(* LS Electric XG5000 project: XEM_Motion_Demo *)
(* PLC LSPLC *)
(* module base 0 slot 0: Input/Output Module:XEM-DN/DP32HP (DC 24V Input, Transistor Output, 32 Contacts) *)
(* module base 0 slot 1: Internal Positioning:XBF-PO06E (Open Collector Type, 6 Axis) *)
VAR_GLOBAL
    Axis1_Command : Motion_Command_type; (* Commands for Axis 1 *)
    Axis1_Status : Motion_Status_type; (* Status for axis 1 *)
    Axis2_Command : Motion_Command_type; (* Commands for Axis 2 *)
    Axis2_Status : Motion_Status_type; (* Status for axis 2 *)
    Axis3_Command : Motion_Command_type; (* Commands for Axis 3 *)
    Axis3_Status : Motion_Status_type; (* Status for axis 3 *)
    Reset_Servo_Errors : BOOL; (* Acknowledge servo errors *)
    Turn_On_Servos : BOOL; (* Command to turn on all the servos *)
END_VAR

TYPE Motion_Command_type : (* contains motion commands and data for those commands *)
STRUCT
    Servo_On : BOOL; (* Command to turn servo on *)
    Home : BOOL; (* command to home axis *)
    Direct_Absolute_Move : BOOL; (* command for direct start absolute move *)
    Direct_Relative_Move : BOOL; (* command for direct start relative move *)
    Direct_Feed_Move : BOOL; (* command to perform a direct start feed move *)
    Direct_Speed_Move : BOOL; (* command to run axis direct start speed control. *)
    Indirect_Absolute_Move : BOOL; (* command for indirect start absolute move *)
    Indirect_Relative_Move : BOOL; (* command for indirect start relative move *)
    Indirect_Feed_Move : BOOL; (* command for indirect start feed move *)
    Indirect_Speed_Move : BOOL; (* command for indirect start speed control. *)
    Linear_Interpolation_Move : BOOL; (* command for indirect start for linear interpolation move *)
    Cirular_Interpolation_Start : BOOL; (* command for indirect start of circular interpolation move *)
    Helical_Interpolation_Start : BOOL; (* command for indirect start of helical interpolation move *)
    Ellipse_Interpolation_Start : BOOL; (* command to start ellipse interpolation. *)
    Stop_Axis : BOOL; (* perform a deceleration stop *)
    EStop_Axis : BOOL; (* peform an emergency stop *)
    Reset_Axis_Error : BOOL; (* reset an axis error *)
    Target_Position : DINT; (* target position for direct start moves in pulses *)
    Target_Speed : UDINT; (* target speed for direct start moves in pulses/sec *)
    Dwell_Time : UINT; (* dwell time in milliseconds *)
    Accel_Selection : USINT; (* Acceleration setting in XG-PM settings to use. *)
    Decel_Selection : USINT; (* Deceleration setting in XG-PM settings to use *)
END_STRUCT;
END_TYPE

TYPE Motion_Status_type : (* Motion status information *)
STRUCT
    Axis_Ready : BOOL; (* axis is ready for commands *)
    Busy : BOOL; (* status that the axis is busy *)
    Error_Present : BOOL; (* status of an error *)
    Move_Done : BOOL; (* status that move is done *)
    Homed : BOOL; (* status that axis is homed. *)
    Current_Position_Pulses : DINT; (* Current position of the axis in pulses *)
    Current_Speed_Pulses : DINT; (* Current speed of the axis in pulses *)
    Current_Torque : INT; (* current torque *)
    Error_Number : UINT; (* current error number *)
    Commanded_Position : DINT; (* commanded position *)
    Commanded_Speed : DINT; (* commanded speed *)
    Current_Step_Number : UINT; (* current step number of the operation being performed *)
    State1 : ARRAY[0..7] OF BOOL; (* array for state 1 of Axis state fb *)
    State2 : ARRAY[0..7] OF BOOL; (* array for state 2 of Axis state fb *)
    State3 : ARRAY[0..7] OF BOOL; (* array for state 3 of Axis state fb *)
    State4 : ARRAY[0..7] OF BOOL; (* array for state 4 of Axis state fb *)
    State5 : ARRAY[0..7] OF BOOL; (* array for state 5 of Axis state fb *)
    State6 : ARRAY[0..7] OF BOOL; (* array for state 6 of Axis state fb *)
    State7 : ARRAY[0..7] OF BOOL; (* array for state 7 of Axis state fb *)
    Servo_Drive_Ready : BOOL; (* status that the servo drive being controlled is ready *)
    Servo_Drive_Error : BOOL; (* Status that the servo drive being controlled doesn't have an error *)
END_STRUCT;
END_TYPE

PROGRAM Interpolation_Routines (* task: Scan Program *)
(* control the demo code for interpolation movements *)
VAR
    Axes_Are_Homed : BOOL; (* status that the 3 axes are homed *)
    Axes_Are_Ready : BOOL; (* status command that axes 1 thru 3 are ready *)
    Home_Axes : BOOL; (* home all the axes *)
    Motion_Manager_State : USINT := 0; (* State machine variable for motion manager *)
    Run_Circular_Interpolation : BOOL := 0; (* command to run circular interpolation demo *)
    Run_Ellipse_Interpolation : BOOL := 0; (* Command to run ellipse interpolation demo *)
    Run_Helical_Interpolation : BOOL := 0; (* command to run helical interpolation demo *)
    Run_Linear_Interpolation : BOOL := 0; (* command to run linear interpolation demo *)
    TempInt : INT;
    TempWord : WORD := 60502;
END_VAR
VAR_EXTERNAL
    Axis1_Command : Motion_Command_type; (* Commands for Axis 1 *)
    Axis1_Status : Motion_Status_type; (* Status for axis 1 *)
    Axis2_Command : Motion_Command_type; (* Commands for Axis 2 *)
    Axis2_Status : Motion_Status_type; (* Status for axis 2 *)
    Axis3_Command : Motion_Command_type; (* Commands for Axis 3 *)
    Axis3_Status : Motion_Status_type; (* Status for axis 3 *)
    Turn_On_Servos : BOOL; (* Command to turn on all the servos *)
END_VAR
(* 
AutomationDirect.com has provided this code for convenience. This sample code is provided "as-is" with no expressed or implied warranty. 
 If the end user includes any of the sample code (in whole or part), it is the user's responsibility to completely modify, integrate, and test any code to ensure it meets all system and 
 safety requirements for the intended application or system.
 *)


//Make sure axes are ready for commands
IF (Axis1_Status.Axis_Ready AND Axis2_Status.Axis_Ready AND Axis3_Status.Axis_Ready) AND (Axis1_Status.Busy = FALSE) AND (Axis2_Status.Busy = FALSE) AND (Axis3_Status.Busy = FALSE) THEN
	Axes_Are_Ready := TRUE;
ELSE
	Axes_Are_Ready := FALSE;

END_IF;
	
//make sure Axes are homed
IF Axis1_Status.Homed AND Axis2_Status.Homed AND Axis3_Status.Homed THEN
	Axes_Are_Homed := TRUE;
ELSE	
	Axes_Are_Homed := FALSE;
	
END_IF;

//Reset State machine if there is a drive alarm or the servos are turned off.
IF (%IX0.0.11 = FALSE) OR (Turn_On_Servos = FALSE) THEN
	Motion_Manager_State := 0;
END_IF;

(* State machine for running the three interpolation demos.  It will move axes to starting positions using the direct start commands of those axes. *)
CASE Motion_Manager_State OF
	
	//wait for command to run a demo.
	0:
		Axis1_Command.Direct_Absolute_Move := FALSE;
		Axis2_Command.Direct_Absolute_Move := FALSE;
		Axis3_Command.Direct_Absolute_Move := FALSE;
		
		//home axes 
		IF Axes_Are_Ready AND Home_Axes THEN
			Home_Axes := FALSE;
			Motion_Manager_State := 100;
			
		//Allow interpolation commands if axes are ready and homed.  They use absolute movements to go to starting positions	
		ELSIF Axes_Are_Ready AND Axes_Are_Homed THEN
			
				IF (Run_Linear_Interpolation = TRUE) THEN
					Run_Linear_Interpolation := FALSE;
					Motion_Manager_State := 10;
				
				ELSIF(Run_Circular_Interpolation = TRUE) THEN
					Run_Circular_Interpolation := FALSE;
					Motion_Manager_State := 20;
					
				ELSIF(Run_Helical_Interpolation = TRUE) THEN
					Run_Helical_Interpolation := FALSE;
					Motion_Manager_State := 30;		
					
				ELSIF(Run_Ellipse_Interpolation = TRUE) THEN
					Run_Ellipse_Interpolation := FALSE;
					Motion_Manager_State := 40;	
						
				END_IF;	

		
		//Reset Interpolation commands if axes are not ready
		ELSE	
				Run_Helical_Interpolation := FALSE;
				Run_Circular_Interpolation := FALSE;
				Run_Linear_Interpolation := FALSE;
		END_IF;
	
	
	(**********************
	     Peform Linear interpolation.
	     ***************************) 
	// Move Axis 3(z on gantry) up so that Axis 1(x) and Axis 2(y) can be moved to starting position.			
	10:	
		IF (Axis3_Status.Current_Position_Pulses = 200)  THEN
			Motion_Manager_State := 11;
			
		ELSE	
			Axis3_Command.Target_Position :=  200;
			Axis3_Command.Target_Speed := 500;
			
			Axis3_Command.Direct_Absolute_Move := TRUE;
			
			IF(Axis3_Status.Current_Position_Pulses = 200) THEN
				Axis3_Command.Direct_Absolute_Move := FALSE;
				Motion_Manager_State := 11;
			END_IF;
			
		END_IF;	
		
	//Axis 1 (x) and Axis 2(y) can move to linear interpolation start position	
	11: 
		Axis1_Command.Target_Position :=  200;
		Axis1_Command.Target_Speed := 500;		
			
		Axis2_Command.Target_Position :=  200;
		Axis2_Command.Target_Speed := 500;
		
		Axis1_Command.Direct_Absolute_Move := TRUE;
		Axis2_Command.Direct_Absolute_Move := TRUE;
	
		
		IF (Axis1_Status.Current_Position_Pulses = 200)  AND (Axis2_Status.Current_Position_Pulses = 200) THEN
			Axis1_Command.Direct_Absolute_Move := FALSE;
			Axis2_Command.Direct_Absolute_Move := FALSE;
			Axis3_Command.Direct_Absolute_Move := FALSE;
			Motion_Manager_State := 12;
		END_IF;	
		
	// Move Axis 3 (z) to 0 position so pen is touching paper	
	12:	
		Axis3_Command.Target_Position :=  0;
		Axis3_Command.Target_Speed := 500;
		
		Axis3_Command.Direct_Absolute_Move := TRUE;
	
		
		IF(Axis3_Status.Current_Position_Pulses = 0) THEN
			Axis3_Command.Direct_Absolute_Move := FALSE;
			Motion_Manager_State := 13;
		END_IF;

	//Start linear interpolation command. Axis 1 is master so it is the only XPM_IST that needs to be run
	13:
		IF Axis1_Status.Axis_Ready AND Axis2_Status.Axis_Ready THEN
			Axis1_Command.Linear_Interpolation_Move := TRUE;
		END_IF;	
		
	 	IF (Axis1_Status.Busy = TRUE)  AND (Axis2_Status.Busy = TRUE) THEN
			Motion_Manager_State := 14;
		END_IF;	
		
	//wait for interpolation to be done then go back to wait for command state	
	14:
		IF Axis1_Status.Move_Done AND Axis2_Status.Move_Done THEN
			Motion_Manager_State := 15;
		END_IF;
		
	//Move the axes to a wait position	 for states 15 and 16
	15:	
			Axis3_Command.Target_Position :=  200;
			Axis3_Command.Target_Speed := 500;			
			Axis3_Command.Direct_Absolute_Move := TRUE;
			
			IF(Axis3_Status.Current_Position_Pulses = 200) THEN
				Axis3_Command.Direct_Absolute_Move := FALSE;
				Motion_Manager_State := 16;
			END_IF;
		
	16:
		Axis1_Command.Target_Position :=  0;
		Axis1_Command.Target_Speed := 500;		
			
		Axis2_Command.Target_Position :=  0;
		Axis2_Command.Target_Speed := 500;
		
		Axis1_Command.Direct_Absolute_Move := TRUE;
		Axis2_Command.Direct_Absolute_Move := TRUE;		
	
		IF (Axis1_Status.Current_Position_Pulses = 0)  AND (Axis2_Status.Current_Position_Pulses = 0) THEN
			Axis1_Command.Direct_Absolute_Move := FALSE;
			Axis2_Command.Direct_Absolute_Move := FALSE;
			Axis3_Command.Direct_Absolute_Move := FALSE;
			Motion_Manager_State := 0;
		END_IF;	
	
	
	(******************************
		 Peform Circular interpolation. 
		 **********************)
	 //MOVE Axis 3(z on gantry) up so that Axis 1(x) and Axis 2(y) can be moved to starting position.			
	20:	
		
		IF (Axis3_Status.Current_Position_Pulses = 200)   THEN
			Motion_Manager_State := 21;
			
		ELSE	
			Axis3_Command.Target_Position :=  200;
			Axis3_Command.Target_Speed := 500;
			
			Axis3_Command.Direct_Absolute_Move := TRUE;
			
			IF(Axis3_Status.Current_Position_Pulses = 200) THEN
				Axis3_Command.Direct_Absolute_Move := FALSE;
				Motion_Manager_State := 21;
			END_IF;
			
		END_IF;	
		
	// Axis 1 (x) and Axis 2(y) can move to circular interpolation start position	
	21: 
		Axis1_Command.Target_Position :=  200;
		Axis1_Command.Target_Speed := 500;		
			
		Axis2_Command.Target_Position :=  1500;
		Axis2_Command.Target_Speed := 500;
		
		Axis1_Command.Direct_Absolute_Move := TRUE;
		Axis2_Command.Direct_Absolute_Move := TRUE;
	
		
		IF (Axis1_Status.Current_Position_Pulses = 200)  AND (Axis2_Status.Current_Position_Pulses = 1500) THEN
			Axis1_Command.Direct_Absolute_Move := FALSE;
			Axis2_Command.Direct_Absolute_Move := FALSE;
			Axis3_Command.Direct_Absolute_Move := FALSE;
			Motion_Manager_State := 22;
		END_IF;	
		
	// move Axis 3 (z) to 0 position so pen is touching paper	
	22:	
		Axis3_Command.Target_Position :=  0;
		Axis3_Command.Target_Speed := 500;
		
		Axis3_Command.Direct_Absolute_Move := TRUE;
	
		
		IF(Axis3_Status.Current_Position_Pulses = 0) THEN
			Axis3_Command.Direct_Absolute_Move := FALSE;
			Motion_Manager_State := 23;
		END_IF;
	
	//Start Circular interpolation command. Axis 1 is master so it is the only XPM_IST that needs to be run
	23:
		IF Axis1_Status.Axis_Ready AND Axis2_Status.Axis_Ready THEN
			Axis1_Command.Cirular_Interpolation_Start := TRUE;
		END_IF;	

	 	IF (Axis1_Status.Busy = TRUE)  AND (Axis2_Status.Busy = TRUE) THEN
			Motion_Manager_State := 24;
		END_IF;			
	
	//wait for interpolation to be done 
	24:
		IF Axis1_Status.Move_Done AND Axis2_Status.Move_Done THEN
			Motion_Manager_State := 25;
		END_IF;	
	
		//Move the axes to a wait position	 for states 25 and 26
	25:	
			Axis3_Command.Target_Position :=  200;
			Axis3_Command.Target_Speed := 500;			
			Axis3_Command.Direct_Absolute_Move := TRUE;
			
			IF(Axis3_Status.Current_Position_Pulses = 200) THEN
				Axis3_Command.Direct_Absolute_Move := FALSE;
				Motion_Manager_State := 26;
			END_IF;
		
	26:
		Axis1_Command.Target_Position :=  0;
		Axis1_Command.Target_Speed := 500;		
			
		Axis2_Command.Target_Position :=  0;
		Axis2_Command.Target_Speed := 500;
		
		Axis1_Command.Direct_Absolute_Move := TRUE;
		Axis2_Command.Direct_Absolute_Move := TRUE;		
	
		IF (Axis1_Status.Current_Position_Pulses = 0)  AND (Axis2_Status.Current_Position_Pulses = 0) THEN
			Axis1_Command.Direct_Absolute_Move := FALSE;
			Axis2_Command.Direct_Absolute_Move := FALSE;
			Axis3_Command.Direct_Absolute_Move := FALSE;
			Motion_Manager_State := 0;
		END_IF;	
	
	
(******************************
		 Peform Helical interpolation. 
		 **********************)
	 //MOVE Axis 3(z on gantry) up so that Axis 1(x) and Axis 2(y) can be moved to starting position.			
	30:	
		
		IF (Axis3_Status.Current_Position_Pulses = 200)   THEN
			Motion_Manager_State := 31;
			
		ELSE	
			Axis3_Command.Target_Position :=  200;
			Axis3_Command.Target_Speed := 500;
			
			Axis3_Command.Direct_Absolute_Move := TRUE;
			
			IF(Axis3_Status.Current_Position_Pulses = 200) THEN
				Axis3_Command.Direct_Absolute_Move := FALSE;
				Motion_Manager_State := 31;
			END_IF;
			
		END_IF;	
		
	// Axis 1 (x) and Axis 2(y) can move to helical interpolation start position	
	31: 
		Axis1_Command.Target_Position :=  600;
		Axis1_Command.Target_Speed := 500;		
			
		Axis2_Command.Target_Position :=  400;
		Axis2_Command.Target_Speed := 500;
		
		Axis1_Command.Direct_Absolute_Move := TRUE;
		Axis2_Command.Direct_Absolute_Move := TRUE;
	
		
		IF (Axis1_Status.Current_Position_Pulses = 600)  AND (Axis2_Status.Current_Position_Pulses = 400) THEN
			Axis1_Command.Direct_Absolute_Move := FALSE;
			Axis2_Command.Direct_Absolute_Move := FALSE;
			Axis3_Command.Direct_Absolute_Move := FALSE;
			Motion_Manager_State := 32;
		END_IF;	
		
	// move Axis 3 (z) to 0 position so pen is touching paper	
	32:	
		Axis3_Command.Target_Position :=  0;
		Axis3_Command.Target_Speed := 500;
		
		Axis3_Command.Direct_Absolute_Move := TRUE;
	
		
		IF(Axis3_Status.Current_Position_Pulses = 0) THEN
			Axis3_Command.Direct_Absolute_Move := FALSE;
			Motion_Manager_State := 33;
		END_IF;
	
	//Start Helical interpolation command. Axis 1 is master so it is the only XPM_IST that needs to be run
	33:
		IF Axis1_Status.Axis_Ready AND Axis2_Status.Axis_Ready AND Axis3_Status.Axis_Ready THEN
			Axis1_Command.Helical_Interpolation_Start := TRUE;
		END_IF;	

	 	IF (Axis1_Status.Busy = TRUE)  AND (Axis2_Status.Busy = TRUE) AND (Axis3_Status.Busy = TRUE) THEN
			Motion_Manager_State := 34;
		END_IF;	
		
	//wait for interpolation to be done 
	34:
		IF Axis1_Status.Move_Done AND Axis2_Status.Move_Done THEN
			Motion_Manager_State := 35;
		END_IF;	
	
		//Move the axes to a wait position for states 35 and 36
	35:	
			Axis3_Command.Target_Position :=  200;
			Axis3_Command.Target_Speed := 500;			
			Axis3_Command.Direct_Absolute_Move := TRUE;
			
			IF(Axis3_Status.Current_Position_Pulses = 200) THEN
				Axis3_Command.Direct_Absolute_Move := FALSE;
				Motion_Manager_State := 36;
			END_IF;
		
	36:
		Axis1_Command.Target_Position :=  0;
		Axis1_Command.Target_Speed := 100;		
			
		Axis2_Command.Target_Position :=  0;
		Axis2_Command.Target_Speed := 500;
		
		Axis1_Command.Direct_Absolute_Move := TRUE;
		Axis2_Command.Direct_Absolute_Move := TRUE;		
	
		IF (Axis1_Status.Current_Position_Pulses = 0)  AND (Axis2_Status.Current_Position_Pulses = 0) THEN
			Axis1_Command.Direct_Absolute_Move := FALSE;
			Axis2_Command.Direct_Absolute_Move := FALSE;
			Axis3_Command.Direct_Absolute_Move := FALSE;
			Motion_Manager_State := 0;
		END_IF;		
	
	
	
(******************************
		 Peform Ellipse interpolation. 
		 **********************)
	 //MOVE Axis 3(z on gantry) up so that Axis 1(x) and Axis 2(y) can be moved to starting position.			
	40:	
		
		IF (Axis3_Status.Current_Position_Pulses = 200)   THEN
			Motion_Manager_State := 41;
			
		ELSE	
			Axis3_Command.Target_Position :=  200;
			Axis3_Command.Target_Speed := 500;
			
			Axis3_Command.Direct_Absolute_Move := TRUE;
			
			IF(Axis3_Status.Current_Position_Pulses = 200) THEN
				Axis3_Command.Direct_Absolute_Move := FALSE;
				Motion_Manager_State := 41;
			END_IF;
			
		END_IF;	
		
	//Axis 1 (x) and Axis 2(y) can move to ellipse interpolation start position	
	41: 
		Axis1_Command.Target_Position :=  0;
		Axis1_Command.Target_Speed := 500;		
			
		Axis2_Command.Target_Position :=  0;
		Axis2_Command.Target_Speed := 500;
		
		Axis1_Command.Direct_Absolute_Move := TRUE;
		Axis2_Command.Direct_Absolute_Move := TRUE;
	
		
		IF (Axis1_Status.Current_Position_Pulses = 0)  AND (Axis2_Status.Current_Position_Pulses = 0) THEN
			Axis1_Command.Direct_Absolute_Move := FALSE;
			Axis2_Command.Direct_Absolute_Move := FALSE;
			Axis3_Command.Direct_Absolute_Move := FALSE;
			Motion_Manager_State := 42;
		END_IF;	
		
	// move Axis 3 (z) to 0 position so pen is touching paper	
	42:	
		Axis3_Command.Target_Position :=  0;
		Axis3_Command.Target_Speed := 500;
		
		Axis3_Command.Direct_Absolute_Move := TRUE;
	
		
		IF(Axis3_Status.Current_Position_Pulses = 0) THEN
			Axis3_Command.Direct_Absolute_Move := FALSE;
			Motion_Manager_State := 43;
		END_IF;
	
	//Start Ellipse interpolation command. Axis 1 is master so it is the only XPM_ELIN that needs to be run
	43:
		IF Axis1_Status.Axis_Ready AND Axis2_Status.Axis_Ready THEN
			Axis1_Command.Ellipse_Interpolation_Start := TRUE;
		END_IF;	

	 	IF (Axis1_Status.Busy = TRUE)  AND (Axis2_Status.Busy = TRUE) THEN
			Motion_Manager_State := 44;
		END_IF;			
	
	//wait for interpolation to be done 
	44:
		IF Axis1_Status.Move_Done AND Axis2_Status.Move_Done THEN
			Motion_Manager_State := 45;
		END_IF;	
	
		//Move the axes to a wait position	 for states 45 and 46
	45:	
			Axis3_Command.Target_Position :=  200;
			Axis3_Command.Target_Speed := 500;			
			Axis3_Command.Direct_Absolute_Move := TRUE;
			
			IF(Axis3_Status.Current_Position_Pulses = 200) THEN
				Axis3_Command.Direct_Absolute_Move := FALSE;
				Motion_Manager_State := 46;
			END_IF;
		
	46:
		Axis1_Command.Target_Position :=  0;
		Axis1_Command.Target_Speed := 500;		
			
		Axis2_Command.Target_Position :=  0;
		Axis2_Command.Target_Speed := 500;
		
		Axis1_Command.Direct_Absolute_Move := TRUE;
		Axis2_Command.Direct_Absolute_Move := TRUE;		
	
		IF (Axis1_Status.Current_Position_Pulses = 0)  AND (Axis2_Status.Current_Position_Pulses = 0) THEN
			Axis1_Command.Direct_Absolute_Move := FALSE;
			Axis2_Command.Direct_Absolute_Move := FALSE;
			Axis3_Command.Direct_Absolute_Move := FALSE;
			Motion_Manager_State := 0;
		END_IF;		
	
	
	
	
	//home axes
	100:
		Axis1_Command.Home := TRUE;
		Axis2_Command.Home := TRUE;
		
		IF (Axis1_Status.Homed AND Axis2_Status.Homed) THEN
			Motion_Manager_State := 101;
		END_IF;
	
	//Home Axis 3 separately so the pen doesn't drag on the surface.
	101:
		Axis3_Command.Home := TRUE;
	
		IF (Axis3_Status.Homed) THEN
			Motion_Manager_State := 102;
		END_IF;
 
	//move Axis 3 to a wait position so Pen isn't constantly in contact with the surface
	102:	
			Axis3_Command.Target_Position :=  200;
			Axis3_Command.Target_Speed := 500;			
			Axis3_Command.Direct_Absolute_Move := TRUE;
			
			IF(Axis3_Status.Current_Position_Pulses = 200) THEN
				Axis3_Command.Direct_Absolute_Move := FALSE;
				Motion_Manager_State := 0;
			END_IF;
		
		
END_CASE;
END_PROGRAM

PROGRAM Axis1_Motion_Program (* task: Scan Program *)
(* program for XPM function blocks that perform actions for axis 1 *)
VAR_EXTERNAL
    Axis1_Command : Motion_Command_type; (* Commands for Axis 1 *)
    Axis1_Status : Motion_Status_type; (* Status for axis 1 *)
END_VAR
VAR
    Axis_State_FB : XPM_SRD; (* Axis state function block *)
    Axis_Status_FB : XPM_CRD; (* Axis status function block *)
    CurPos_Conversion_Value : REAL; (* value to convert pulse position to engineering unit position *)
    Deceleration_Stop_FB : XPM_STP; (* function block for deceleration stop *)
    DirectStart_ABS_INC : BOOL; (* False - Absolute Positioning;  True -  Relative Positioning *)
    DirectStart_Control : USINT; (* Control Method for Direct Start.  0 - Position Control; 1 - Speed Control;  2 - FEED Control *)
    Direct_Start_FB : XPM_DST; (* function block for direct start commands *)
    Emergency_Stop_FB : XPM_EMG; (* function block to perform emergency stop *)
    Error_Reset_FB : XPM_RST; (* function block for resetting axis error *)
    Home_FB : XPM_ORG; (* function block to home axis *)
    Indirect_Start_FB : XPM_IST; (* function block to perform indirect start procedures *)
    Indirect_Step_Number : UINT; (* Step number for Indirect movement *)
    TempR1 : REAL; (* temporary real storage *)
    TempR2 : REAL; (* temporary real storage *)
    XPM_ELIN_INST : XPM_ELIN;
END_VAR
VAR
    _e1 : R_TRIG;
    _e2 : R_TRIG;
    _e3 : R_TRIG;
    _e4 : R_TRIG;
    _e5 : R_TRIG;
    _e6 : R_TRIG;
    _e7 : R_TRIG;
    _e8 : R_TRIG;
    _e9 : R_TRIG;
    _e10 : R_TRIG;
    _e11 : R_TRIG;
    _e12 : R_TRIG;
    _e13 : R_TRIG;
    _e14 : R_TRIG;
    _e15 : R_TRIG;
END_VAR

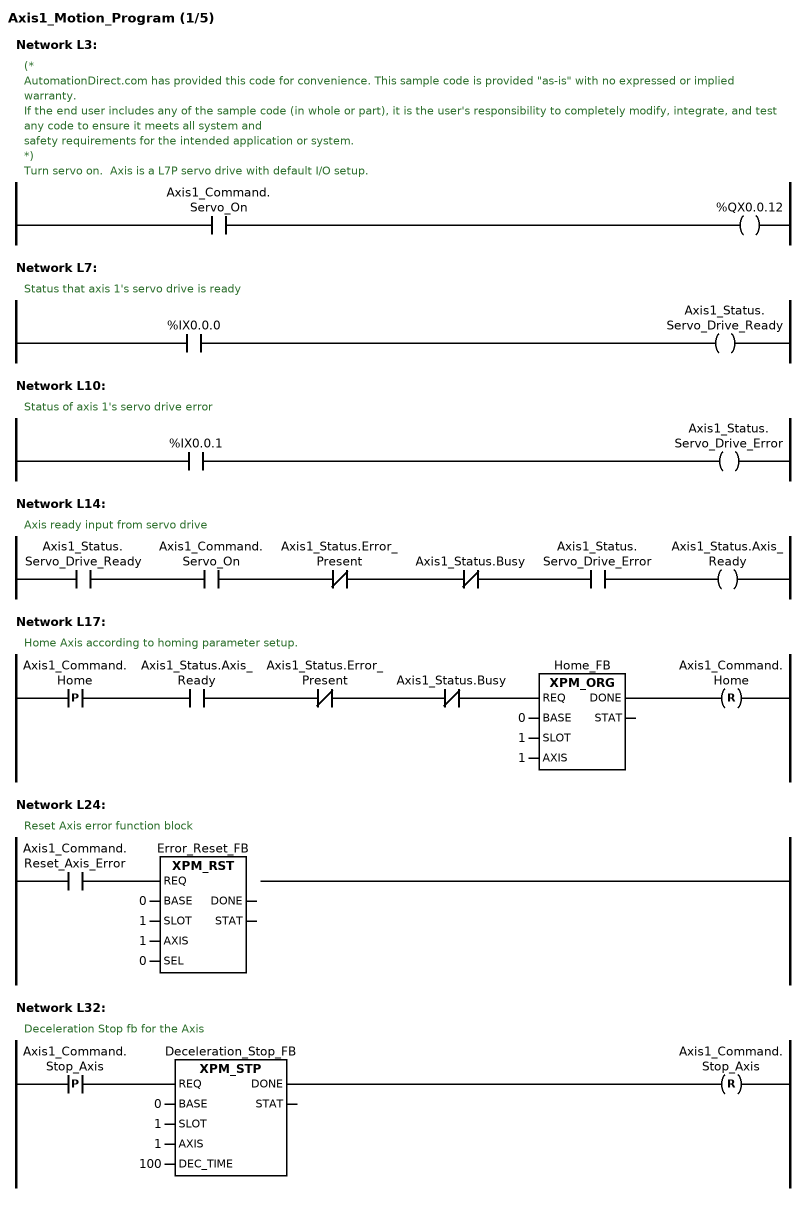
(* ( * / AutomationDirect.com has provided this code for convenience. This sample code is provided "as-is" with no expressed or implied warranty. / If the end user includes any of the sample code (in whole or part), it is the user's responsibility to completely modify, integrate, and test any code to ensure it meets all system and / safety requirements for the intended application or system. / * ) *)
(* Turn servo on.  Axis is a L7P servo drive with default I/O setup. *)
(* Rung L3 *)
%QX0.0.12 := Axis1_Command.Servo_On;
(* Status that axis 1's servo drive is ready *)
(* Rung L7 *)
Axis1_Status.Servo_Drive_Ready := %IX0.0.0;
(* Status of axis 1's servo drive error *)
(* Rung L10 *)
Axis1_Status.Servo_Drive_Error := %IX0.0.1;
(* Axis ready input from servo drive *)
(* Rung L14 *)
Axis1_Status.Axis_Ready := Axis1_Status.Servo_Drive_Ready AND Axis1_Command.Servo_On AND NOT Axis1_Status.Error_Present AND NOT Axis1_Status.Busy AND Axis1_Status.Servo_Drive_Error;
(* Home Axis according to homing parameter setup. *)
(* Rung L17 *)
_e1(CLK := Axis1_Command.Home);
Home_FB(REQ := _e1.Q AND Axis1_Status.Axis_Ready AND NOT Axis1_Status.Error_Present AND NOT Axis1_Status.Busy, BASE := 0, SLOT := 1, AXIS := 1);
IF Home_FB.DONE THEN Axis1_Command.Home := FALSE; END_IF;
(* Reset Axis error function block *)
(* Rung L24 *)
Error_Reset_FB(REQ := Axis1_Command.Reset_Axis_Error, BASE := 0, SLOT := 1, AXIS := 1, SEL := 0);
(* Deceleration Stop fb for the Axis *)
(* Rung L32 *)
_e2(CLK := Axis1_Command.Stop_Axis);
Deceleration_Stop_FB(REQ := _e2.Q, BASE := 0, SLOT := 1, AXIS := 1, DEC_TIME := 100);
IF Deceleration_Stop_FB.DONE THEN Axis1_Command.Stop_Axis := FALSE; END_IF;

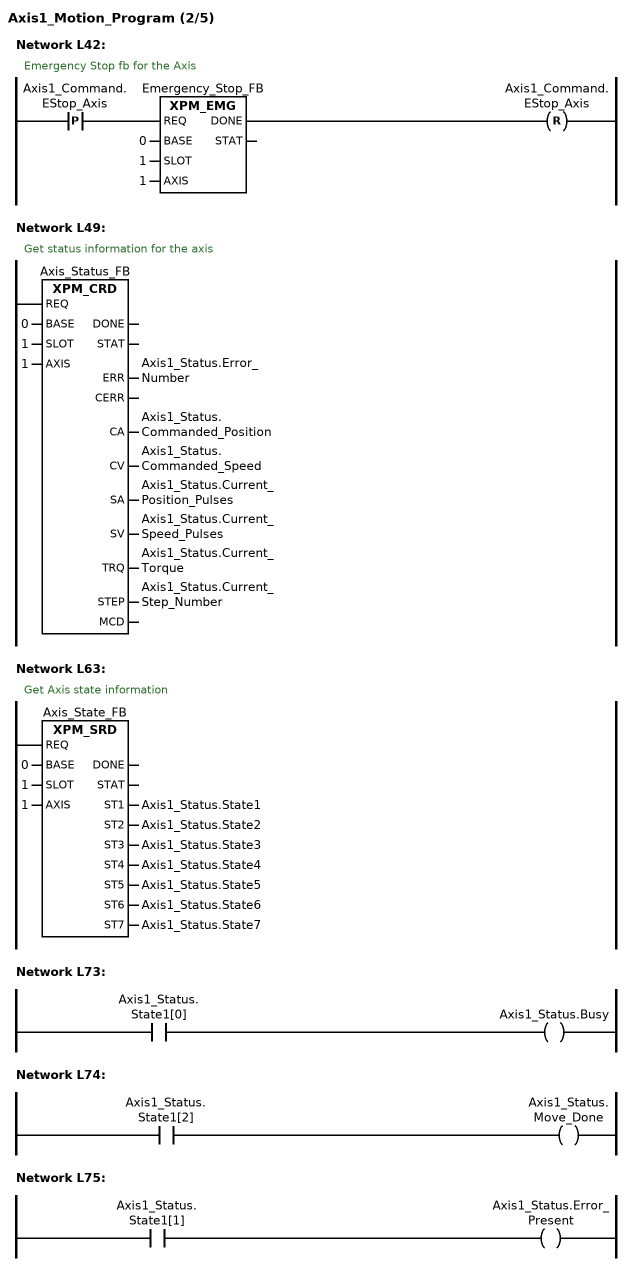
(* Emergency Stop fb for the Axis *)
(* Rung L42 *)
_e3(CLK := Axis1_Command.EStop_Axis);
Emergency_Stop_FB(REQ := _e3.Q, BASE := 0, SLOT := 1, AXIS := 1);
IF Emergency_Stop_FB.DONE THEN Axis1_Command.EStop_Axis := FALSE; END_IF;
(* Get status information for the axis *)
(* Rung L49 *)
Axis_Status_FB(REQ := TRUE, BASE := 0, SLOT := 1, AXIS := 1, ERR => Axis1_Status.Error_Number, CA => Axis1_Status.Commanded_Position, CV => Axis1_Status.Commanded_Speed, SA => Axis1_Status.Current_Position_Pulses, SV => Axis1_Status.Current_Speed_Pulses, TRQ => Axis1_Status.Current_Torque, STEP => Axis1_Status.Current_Step_Number);
(* Get Axis state information *)
(* Rung L63 *)
Axis_State_FB(REQ := TRUE, BASE := 0, SLOT := 1, AXIS := 1, ST1 => Axis1_Status.State1, ST2 => Axis1_Status.State2, ST3 => Axis1_Status.State3, ST4 => Axis1_Status.State4, ST5 => Axis1_Status.State5, ST6 => Axis1_Status.State6, ST7 => Axis1_Status.State7);
(* Rung L73 *)
Axis1_Status.Busy := Axis1_Status.State1[0];
(* Rung L74 *)
Axis1_Status.Move_Done := Axis1_Status.State1[2];
(* Rung L75 *)
Axis1_Status.Error_Present := Axis1_Status.State1[1];

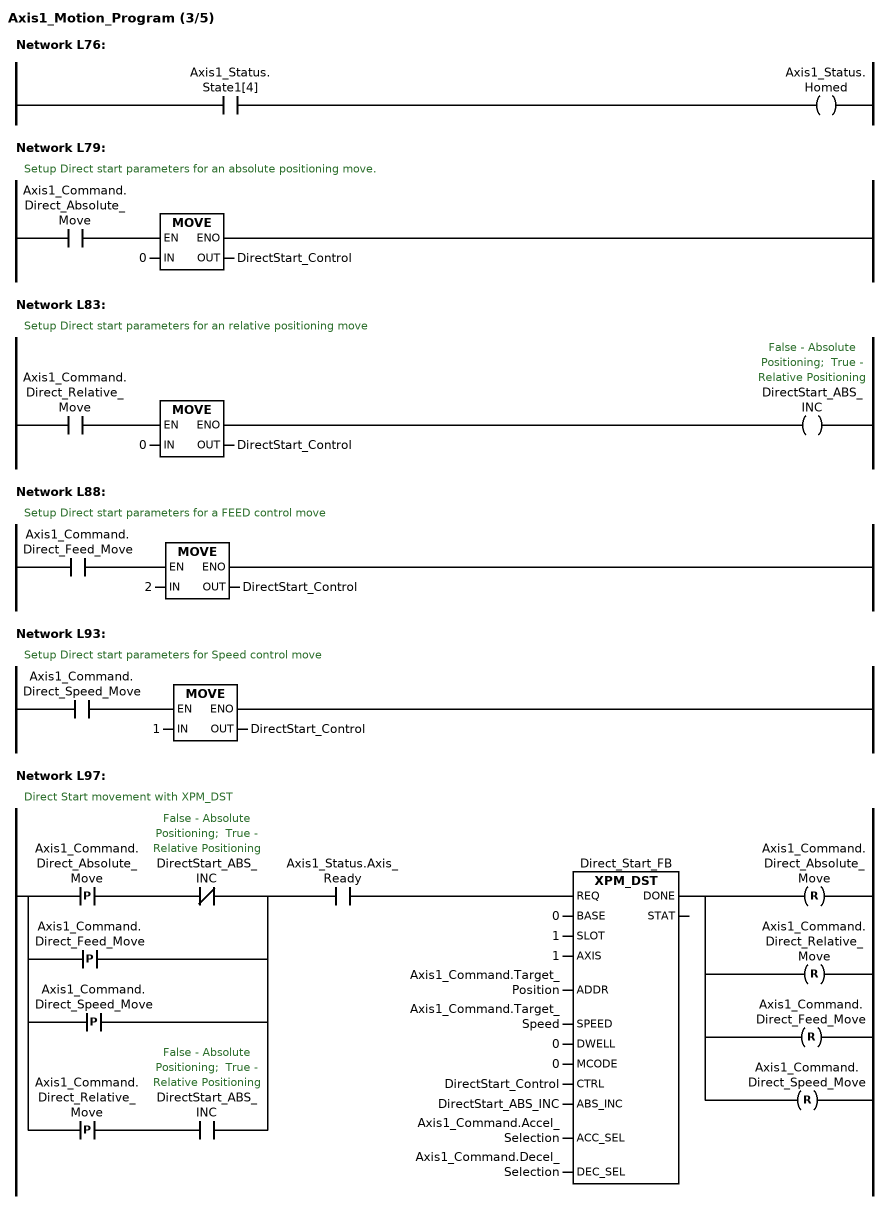
(* Rung L76 *)
Axis1_Status.Homed := Axis1_Status.State1[4];
(* Setup Direct start parameters for an absolute positioning move. *)
(* Rung L79 *)
IF Axis1_Command.Direct_Absolute_Move THEN DirectStart_Control := 0; END_IF;
(* Setup Direct start parameters for an relative positioning move *)
(* Rung L83 *)
IF Axis1_Command.Direct_Relative_Move THEN DirectStart_Control := 0; END_IF;
DirectStart_ABS_INC := Axis1_Command.Direct_Relative_Move;
(* Setup Direct start parameters for a FEED control move *)
(* Rung L88 *)
IF Axis1_Command.Direct_Feed_Move THEN DirectStart_Control := 2; END_IF;
(* Setup Direct start parameters for Speed control move *)
(* Rung L93 *)
IF Axis1_Command.Direct_Speed_Move THEN DirectStart_Control := 1; END_IF;
(* Direct Start movement with XPM_DST *)
(* Rung L97 *)
_e4(CLK := Axis1_Command.Direct_Absolute_Move);
_e5(CLK := Axis1_Command.Direct_Feed_Move);
_e6(CLK := Axis1_Command.Direct_Speed_Move);
_e7(CLK := Axis1_Command.Direct_Relative_Move);
Direct_Start_FB(REQ := ((_e4.Q AND NOT DirectStart_ABS_INC) OR _e5.Q OR _e6.Q OR (_e7.Q AND DirectStart_ABS_INC)) AND Axis1_Status.Axis_Ready, BASE := 0, SLOT := 1, AXIS := 1, ADDR := Axis1_Command.Target_Position, SPEED := Axis1_Command.Target_Speed, DWELL := 0, MCODE := 0, CTRL := DirectStart_Control, ABS_INC := DirectStart_ABS_INC, ACC_SEL := Axis1_Command.Accel_Selection, DEC_SEL := Axis1_Command.Decel_Selection);
IF Direct_Start_FB.DONE THEN
    Axis1_Command.Direct_Absolute_Move := FALSE;
    Axis1_Command.Direct_Relative_Move := FALSE;
    Axis1_Command.Direct_Feed_Move := FALSE;
    Axis1_Command.Direct_Speed_Move := FALSE;
END_IF;

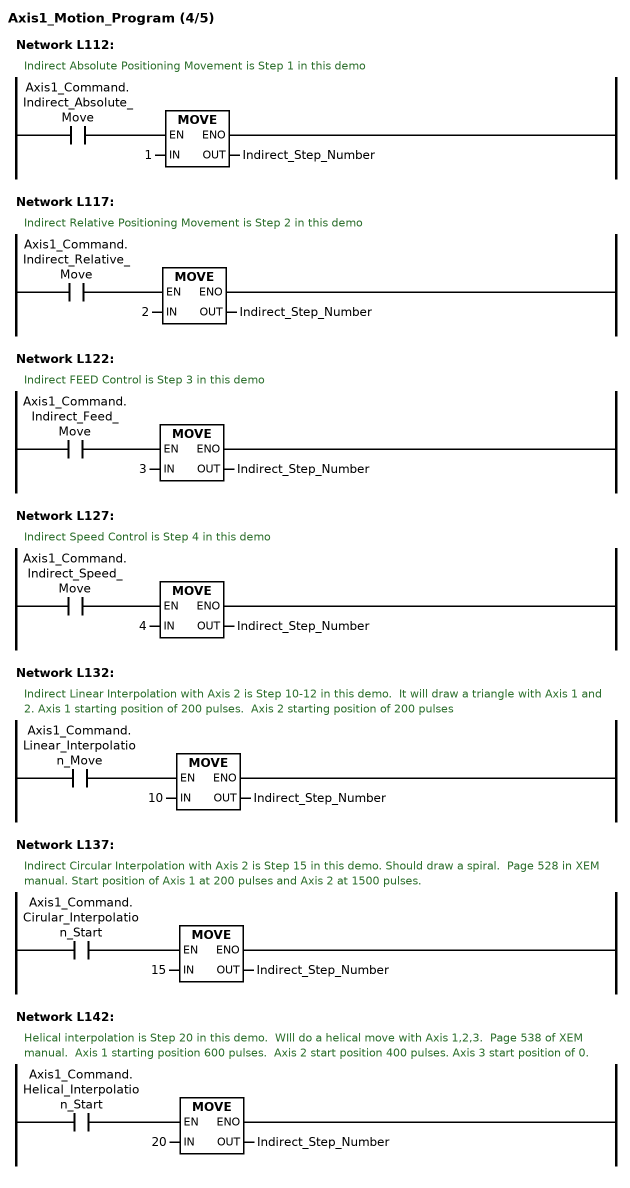
(* Indirect Absolute Positioning Movement is Step 1 in this demo *)
(* Rung L112 *)
IF Axis1_Command.Indirect_Absolute_Move THEN Indirect_Step_Number := 1; END_IF;
(* Indirect Relative Positioning Movement is Step 2 in this demo *)
(* Rung L117 *)
IF Axis1_Command.Indirect_Relative_Move THEN Indirect_Step_Number := 2; END_IF;
(* Indirect FEED Control is Step 3 in this demo *)
(* Rung L122 *)
IF Axis1_Command.Indirect_Feed_Move THEN Indirect_Step_Number := 3; END_IF;
(* Indirect Speed Control is Step 4 in this demo *)
(* Rung L127 *)
IF Axis1_Command.Indirect_Speed_Move THEN Indirect_Step_Number := 4; END_IF;
(* Indirect Linear Interpolation with Axis 2 is Step 10-12 in this demo.  It will draw a triangle with Axis 1 and 2. Axis 1 starting position of 200 pulses.  Axis 2 starting position of 200 pulses *)
(* Rung L132 *)
IF Axis1_Command.Linear_Interpolation_Move THEN Indirect_Step_Number := 10; END_IF;
(* Indirect Circular Interpolation with Axis 2 is Step 15 in this demo. Should draw a spiral.  Page 528 in XEM manual. Start position of Axis 1 at 200 pulses and Axis 2 at 1500 pulses. *)
(* Rung L137 *)
IF Axis1_Command.Cirular_Interpolation_Start THEN Indirect_Step_Number := 15; END_IF;
(* Helical interpolation is Step 20 in this demo.  WIll do a helical move with Axis 1,2,3.  Page 538 of XEM manual.  Axis 1 starting position 600 pulses.  Axis 2 start position 400 pulses. Axis 3 start position of 0. *)
(* Rung L142 *)
IF Axis1_Command.Helical_Interpolation_Start THEN Indirect_Step_Number := 20; END_IF;

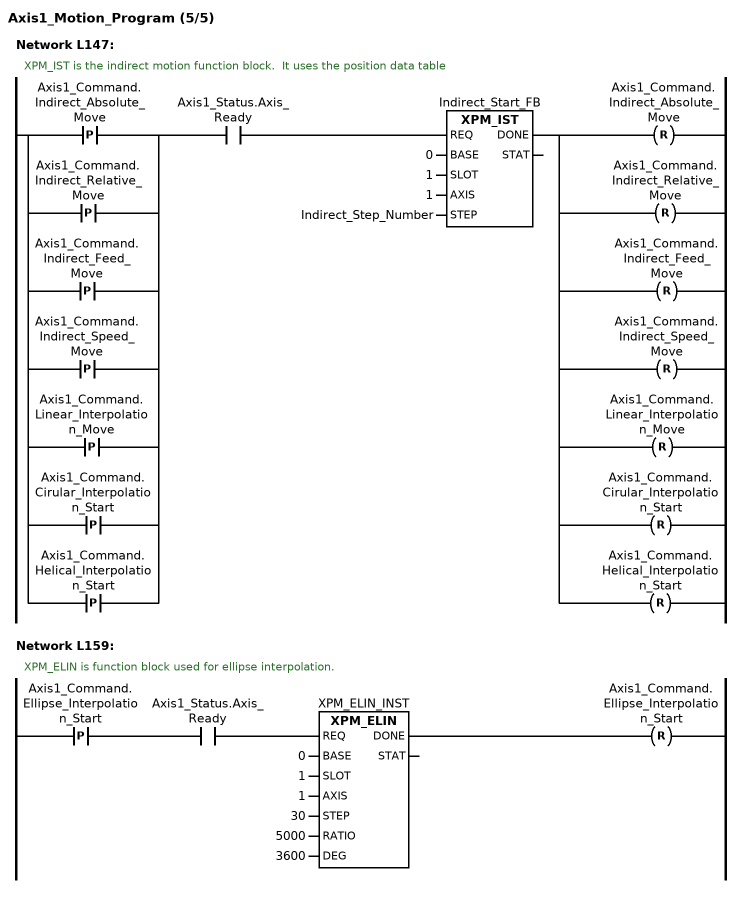
(* XPM_IST is the indirect motion function block.  It uses the position data table *)
(* Rung L147 *)
_e8(CLK := Axis1_Command.Indirect_Absolute_Move);
_e9(CLK := Axis1_Command.Indirect_Relative_Move);
_e10(CLK := Axis1_Command.Indirect_Feed_Move);
_e11(CLK := Axis1_Command.Indirect_Speed_Move);
_e12(CLK := Axis1_Command.Linear_Interpolation_Move);
_e13(CLK := Axis1_Command.Cirular_Interpolation_Start);
_e14(CLK := Axis1_Command.Helical_Interpolation_Start);
Indirect_Start_FB(REQ := (_e8.Q OR _e9.Q OR _e10.Q OR _e11.Q OR _e12.Q OR _e13.Q OR _e14.Q) AND Axis1_Status.Axis_Ready, BASE := 0, SLOT := 1, AXIS := 1, STEP := Indirect_Step_Number);
IF Indirect_Start_FB.DONE THEN
    Axis1_Command.Indirect_Absolute_Move := FALSE;
    Axis1_Command.Indirect_Relative_Move := FALSE;
    Axis1_Command.Indirect_Feed_Move := FALSE;
    Axis1_Command.Indirect_Speed_Move := FALSE;
    Axis1_Command.Linear_Interpolation_Move := FALSE;
    Axis1_Command.Cirular_Interpolation_Start := FALSE;
    Axis1_Command.Helical_Interpolation_Start := FALSE;
END_IF;
(* XPM_ELIN is function block used for ellipse interpolation. *)
(* Rung L159 *)
_e15(CLK := Axis1_Command.Ellipse_Interpolation_Start);
XPM_ELIN_INST(REQ := _e15.Q AND Axis1_Status.Axis_Ready, BASE := 0, SLOT := 1, AXIS := 1, STEP := 30, RATIO := 5000, DEG := 3600);
IF XPM_ELIN_INST.DONE THEN Axis1_Command.Ellipse_Interpolation_Start := FALSE; END_IF;
END_PROGRAM

PROGRAM Axis2_Motion_Program (* task: Scan Program *)
(* program for XPM function blocks that perform actions for axis 2 *)
VAR_EXTERNAL
    Axis2_Command : Motion_Command_type; (* Commands for Axis 2 *)
    Axis2_Status : Motion_Status_type; (* Status for axis 2 *)
END_VAR
VAR
    Axis_State_FB : XPM_SRD; (* Axis state function block *)
    Axis_Status_FB : XPM_CRD; (* Axis status function block *)
    CurPos_Conversion_Value : REAL; (* value to convert pulse position to engineering unit position *)
    Deceleration_Stop_FB : XPM_STP; (* function block for deceleration stop *)
    DirectStart_ABS_INC : BOOL; (* False - Absolute Positioning;  True -  Relative Positioning *)
    DirectStart_Control : USINT; (* Control Method for Direct Start.  0 - Position Control; 1 - Speed Control;  2 - FEED Control *)
    Direct_Start_FB : XPM_DST; (* function block for direct start commands *)
    Emergency_Stop_FB : XPM_EMG; (* function block to perform emergency stop *)
    Error_Reset_FB : XPM_RST; (* function block for resetting axis error *)
    Home_FB : XPM_ORG; (* function block to home axis *)
    Indirect_Start_FB : XPM_IST; (* function block to perform indirect start procedures *)
    Indirect_Step_Number : UINT; (* Step number for Indirect movement *)
    TempR1 : REAL; (* temporary real storage *)
    TempR2 : REAL; (* temporary real storage *)
END_VAR
VAR
    _e1 : R_TRIG;
    _e2 : R_TRIG;
    _e3 : R_TRIG;
    _e4 : R_TRIG;
    _e5 : R_TRIG;
    _e6 : R_TRIG;
    _e7 : R_TRIG;
    _e8 : R_TRIG;
    _e9 : R_TRIG;
    _e10 : R_TRIG;
    _e11 : R_TRIG;
END_VAR

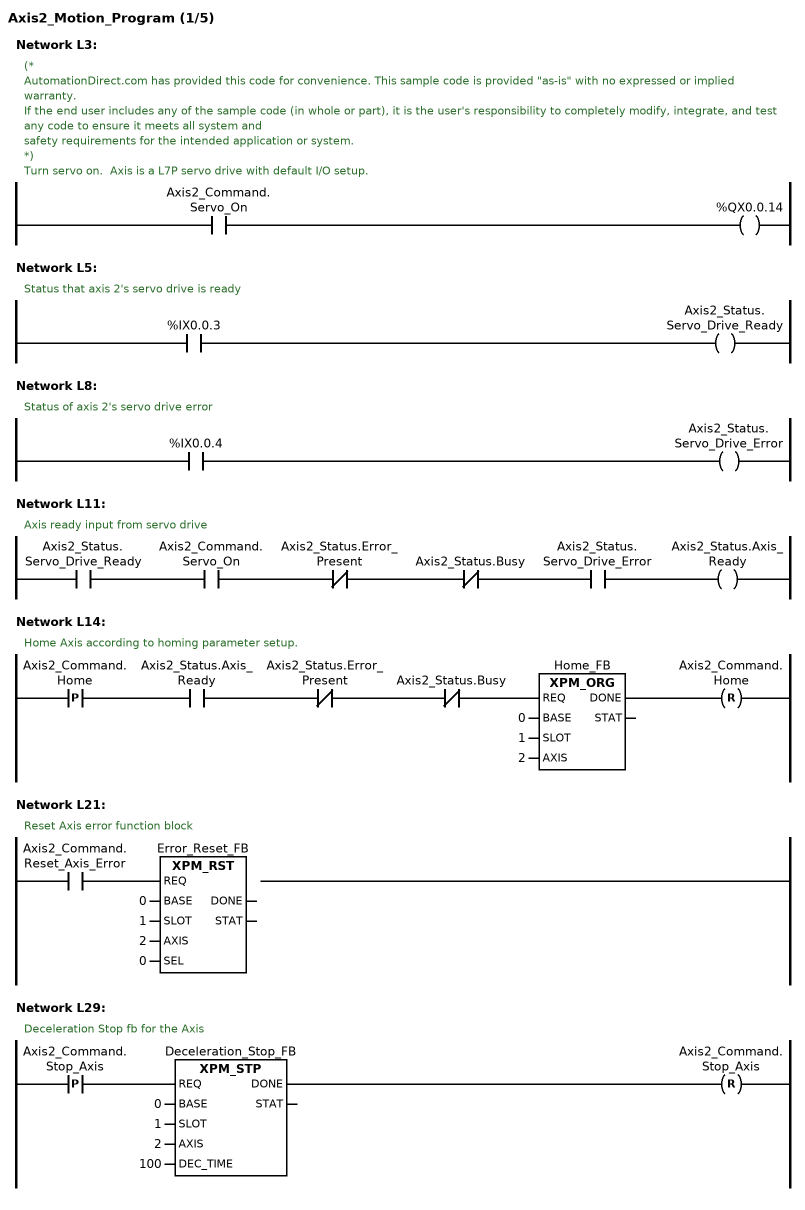
(* ( * / AutomationDirect.com has provided this code for convenience. This sample code is provided "as-is" with no expressed or implied warranty. / If the end user includes any of the sample code (in whole or part), it is the user's responsibility to completely modify, integrate, and test any code to ensure it meets all system and / safety requirements for the intended application or system. / * ) *)
(* Turn servo on.  Axis is a L7P servo drive with default I/O setup. *)
(* Rung L3 *)
%QX0.0.14 := Axis2_Command.Servo_On;
(* Status that axis 2's servo drive is ready *)
(* Rung L5 *)
Axis2_Status.Servo_Drive_Ready := %IX0.0.3;
(* Status of axis 2's servo drive error *)
(* Rung L8 *)
Axis2_Status.Servo_Drive_Error := %IX0.0.4;
(* Axis ready input from servo drive *)
(* Rung L11 *)
Axis2_Status.Axis_Ready := Axis2_Status.Servo_Drive_Ready AND Axis2_Command.Servo_On AND NOT Axis2_Status.Error_Present AND NOT Axis2_Status.Busy AND Axis2_Status.Servo_Drive_Error;
(* Home Axis according to homing parameter setup. *)
(* Rung L14 *)
_e1(CLK := Axis2_Command.Home);
Home_FB(REQ := _e1.Q AND Axis2_Status.Axis_Ready AND NOT Axis2_Status.Error_Present AND NOT Axis2_Status.Busy, BASE := 0, SLOT := 1, AXIS := 2);
IF Home_FB.DONE THEN Axis2_Command.Home := FALSE; END_IF;
(* Reset Axis error function block *)
(* Rung L21 *)
Error_Reset_FB(REQ := Axis2_Command.Reset_Axis_Error, BASE := 0, SLOT := 1, AXIS := 2, SEL := 0);
(* Deceleration Stop fb for the Axis *)
(* Rung L29 *)
_e2(CLK := Axis2_Command.Stop_Axis);
Deceleration_Stop_FB(REQ := _e2.Q, BASE := 0, SLOT := 1, AXIS := 2, DEC_TIME := 100);
IF Deceleration_Stop_FB.DONE THEN Axis2_Command.Stop_Axis := FALSE; END_IF;

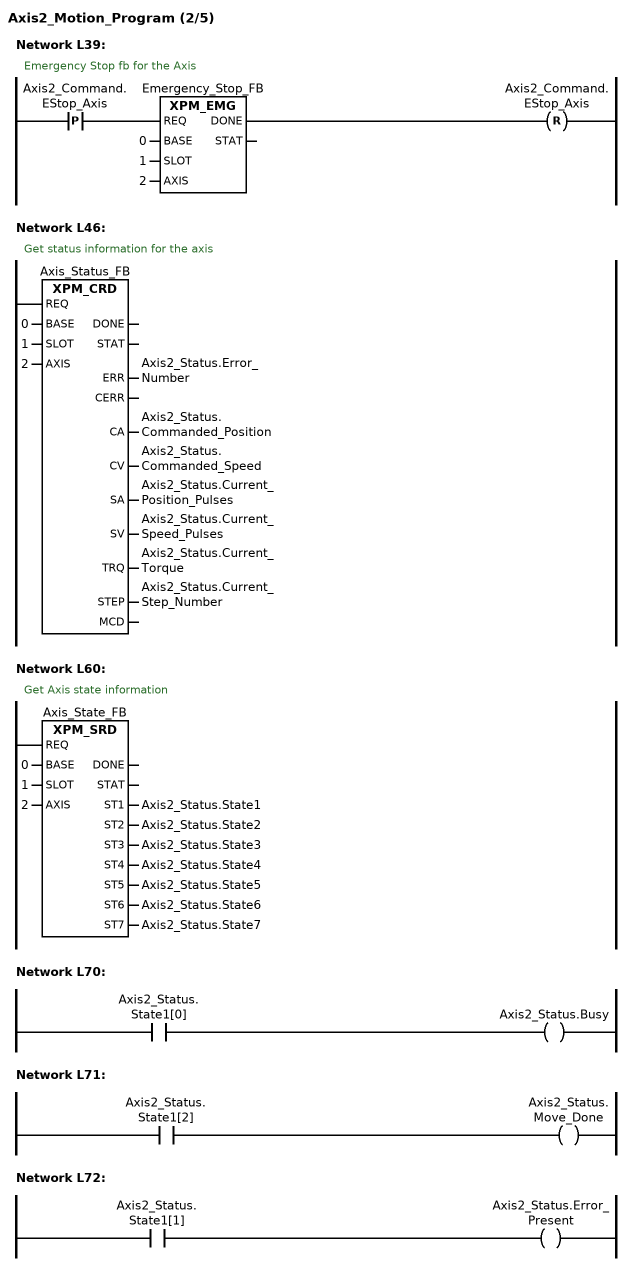
(* Emergency Stop fb for the Axis *)
(* Rung L39 *)
_e3(CLK := Axis2_Command.EStop_Axis);
Emergency_Stop_FB(REQ := _e3.Q, BASE := 0, SLOT := 1, AXIS := 2);
IF Emergency_Stop_FB.DONE THEN Axis2_Command.EStop_Axis := FALSE; END_IF;
(* Get status information for the axis *)
(* Rung L46 *)
Axis_Status_FB(REQ := TRUE, BASE := 0, SLOT := 1, AXIS := 2, ERR => Axis2_Status.Error_Number, CA => Axis2_Status.Commanded_Position, CV => Axis2_Status.Commanded_Speed, SA => Axis2_Status.Current_Position_Pulses, SV => Axis2_Status.Current_Speed_Pulses, TRQ => Axis2_Status.Current_Torque, STEP => Axis2_Status.Current_Step_Number);
(* Get Axis state information *)
(* Rung L60 *)
Axis_State_FB(REQ := TRUE, BASE := 0, SLOT := 1, AXIS := 2, ST1 => Axis2_Status.State1, ST2 => Axis2_Status.State2, ST3 => Axis2_Status.State3, ST4 => Axis2_Status.State4, ST5 => Axis2_Status.State5, ST6 => Axis2_Status.State6, ST7 => Axis2_Status.State7);
(* Rung L70 *)
Axis2_Status.Busy := Axis2_Status.State1[0];
(* Rung L71 *)
Axis2_Status.Move_Done := Axis2_Status.State1[2];
(* Rung L72 *)
Axis2_Status.Error_Present := Axis2_Status.State1[1];

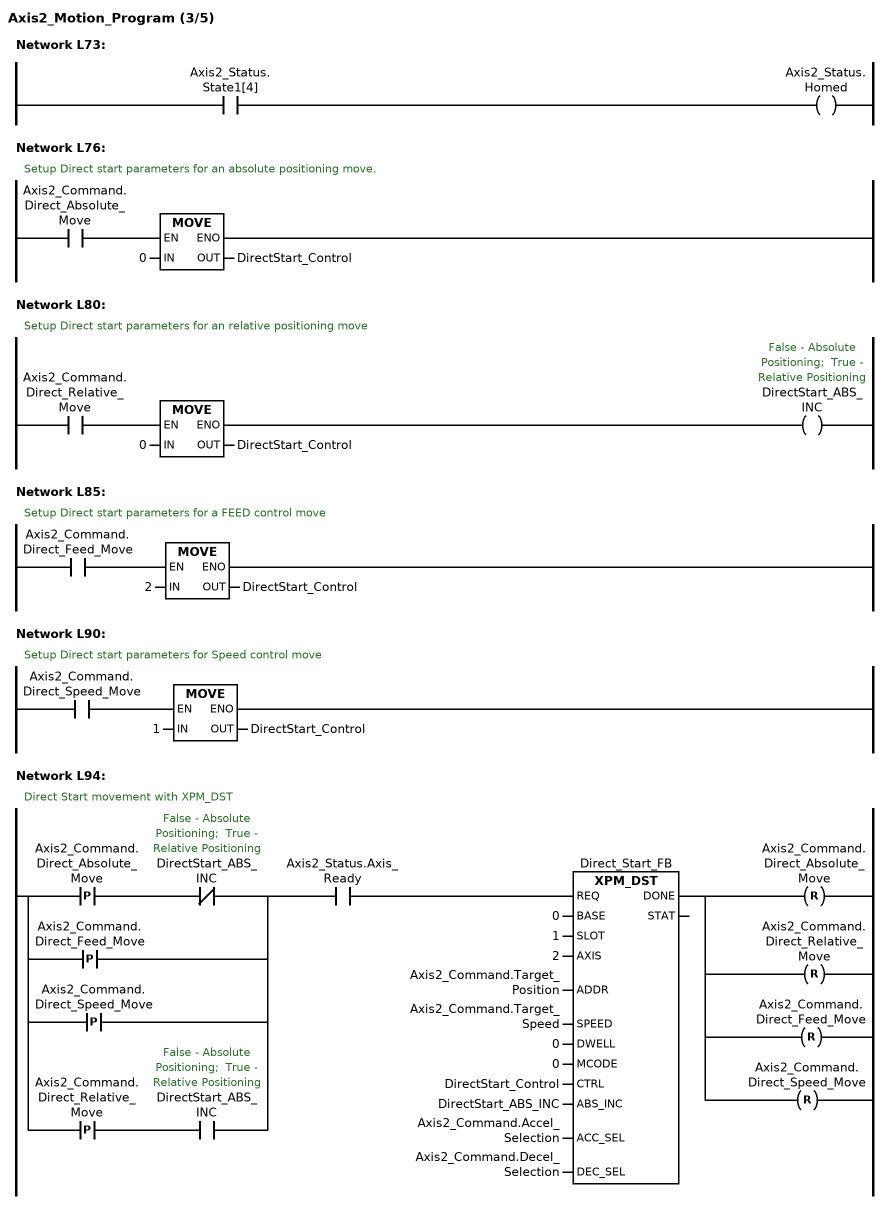
(* Rung L73 *)
Axis2_Status.Homed := Axis2_Status.State1[4];
(* Setup Direct start parameters for an absolute positioning move. *)
(* Rung L76 *)
IF Axis2_Command.Direct_Absolute_Move THEN DirectStart_Control := 0; END_IF;
(* Setup Direct start parameters for an relative positioning move *)
(* Rung L80 *)
IF Axis2_Command.Direct_Relative_Move THEN DirectStart_Control := 0; END_IF;
DirectStart_ABS_INC := Axis2_Command.Direct_Relative_Move;
(* Setup Direct start parameters for a FEED control move *)
(* Rung L85 *)
IF Axis2_Command.Direct_Feed_Move THEN DirectStart_Control := 2; END_IF;
(* Setup Direct start parameters for Speed control move *)
(* Rung L90 *)
IF Axis2_Command.Direct_Speed_Move THEN DirectStart_Control := 1; END_IF;
(* Direct Start movement with XPM_DST *)
(* Rung L94 *)
_e4(CLK := Axis2_Command.Direct_Absolute_Move);
_e5(CLK := Axis2_Command.Direct_Feed_Move);
_e6(CLK := Axis2_Command.Direct_Speed_Move);
_e7(CLK := Axis2_Command.Direct_Relative_Move);
Direct_Start_FB(REQ := ((_e4.Q AND NOT DirectStart_ABS_INC) OR _e5.Q OR _e6.Q OR (_e7.Q AND DirectStart_ABS_INC)) AND Axis2_Status.Axis_Ready, BASE := 0, SLOT := 1, AXIS := 2, ADDR := Axis2_Command.Target_Position, SPEED := Axis2_Command.Target_Speed, DWELL := 0, MCODE := 0, CTRL := DirectStart_Control, ABS_INC := DirectStart_ABS_INC, ACC_SEL := Axis2_Command.Accel_Selection, DEC_SEL := Axis2_Command.Decel_Selection);
IF Direct_Start_FB.DONE THEN
    Axis2_Command.Direct_Absolute_Move := FALSE;
    Axis2_Command.Direct_Relative_Move := FALSE;
    Axis2_Command.Direct_Feed_Move := FALSE;
    Axis2_Command.Direct_Speed_Move := FALSE;
END_IF;

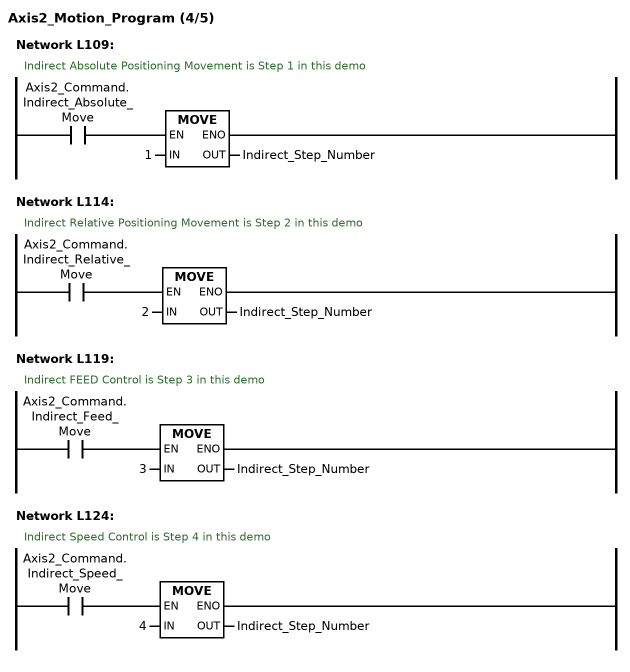
(* Indirect Absolute Positioning Movement is Step 1 in this demo *)
(* Rung L109 *)
IF Axis2_Command.Indirect_Absolute_Move THEN Indirect_Step_Number := 1; END_IF;
(* Indirect Relative Positioning Movement is Step 2 in this demo *)
(* Rung L114 *)
IF Axis2_Command.Indirect_Relative_Move THEN Indirect_Step_Number := 2; END_IF;
(* Indirect FEED Control is Step 3 in this demo *)
(* Rung L119 *)
IF Axis2_Command.Indirect_Feed_Move THEN Indirect_Step_Number := 3; END_IF;
(* Indirect Speed Control is Step 4 in this demo *)
(* Rung L124 *)
IF Axis2_Command.Indirect_Speed_Move THEN Indirect_Step_Number := 4; END_IF;

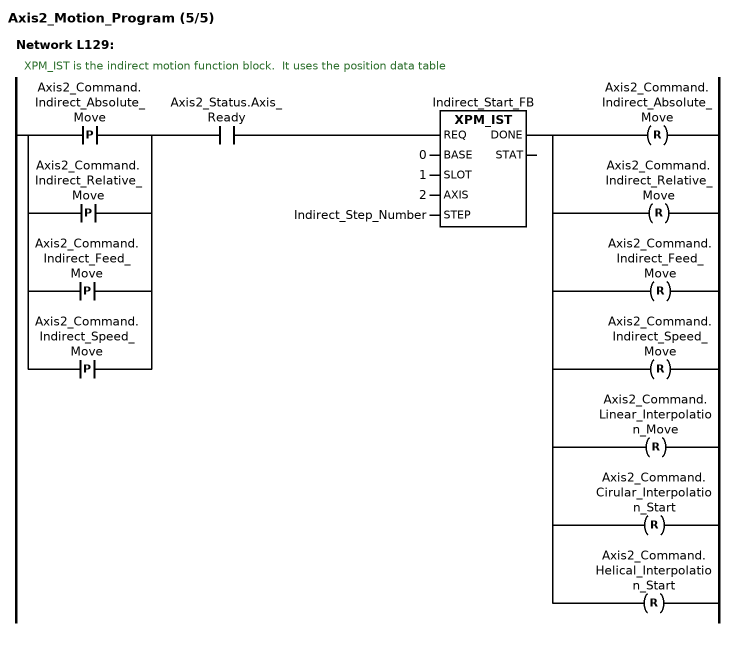
(* XPM_IST is the indirect motion function block.  It uses the position data table *)
(* Rung L129 *)
_e8(CLK := Axis2_Command.Indirect_Absolute_Move);
_e9(CLK := Axis2_Command.Indirect_Relative_Move);
_e10(CLK := Axis2_Command.Indirect_Feed_Move);
_e11(CLK := Axis2_Command.Indirect_Speed_Move);
Indirect_Start_FB(REQ := (_e8.Q OR _e9.Q OR _e10.Q OR _e11.Q) AND Axis2_Status.Axis_Ready, BASE := 0, SLOT := 1, AXIS := 2, STEP := Indirect_Step_Number);
IF Indirect_Start_FB.DONE THEN
    Axis2_Command.Indirect_Absolute_Move := FALSE;
    Axis2_Command.Indirect_Relative_Move := FALSE;
    Axis2_Command.Indirect_Feed_Move := FALSE;
    Axis2_Command.Indirect_Speed_Move := FALSE;
    Axis2_Command.Linear_Interpolation_Move := FALSE;
    Axis2_Command.Cirular_Interpolation_Start := FALSE;
    Axis2_Command.Helical_Interpolation_Start := FALSE;
END_IF;
END_PROGRAM

PROGRAM Axis3_Motion_Program (* task: Scan Program *)
(* program for XPM function blocks that perform actions for axis 3 *)
VAR_EXTERNAL
    Axis3_Command : Motion_Command_type; (* Commands for Axis 3 *)
    Axis3_Status : Motion_Status_type; (* Status for axis 3 *)
END_VAR
VAR
    Axis_State_FB : XPM_SRD; (* Axis state function block *)
    Axis_Status_FB : XPM_CRD; (* Axis status function block *)
    CurPos_Conversion_Value : REAL; (* value to convert pulse position to engineering unit position *)
    Deceleration_Stop_FB : XPM_STP; (* function block for deceleration stop *)
    DirectStart_ABS_INC : BOOL; (* False - Absolute Positioning;  True -  Relative Positioning *)
    DirectStart_Control : USINT; (* Control Method for Direct Start.  0 - Position Control; 1 - Speed Control;  2 - FEED Control *)
    Direct_Start_FB : XPM_DST; (* function block for direct start commands *)
    Emergency_Stop_FB : XPM_EMG; (* function block to perform emergency stop *)
    Error_Reset_FB : XPM_RST; (* function block for resetting axis error *)
    Home_FB : XPM_ORG; (* function block to home axis *)
    Indirect_Start_FB : XPM_IST; (* function block to perform indirect start procedures *)
    Indirect_Step_Number : UINT; (* Step number for Indirect movement *)
    TempR1 : REAL; (* temporary real storage *)
    TempR2 : REAL; (* temporary real storage *)
END_VAR
VAR
    _e1 : R_TRIG;
    _e2 : R_TRIG;
    _e3 : R_TRIG;
    _e4 : R_TRIG;
    _e5 : R_TRIG;
    _e6 : R_TRIG;
    _e7 : R_TRIG;
    _e8 : R_TRIG;
    _e9 : R_TRIG;
    _e10 : R_TRIG;
    _e11 : R_TRIG;
END_VAR

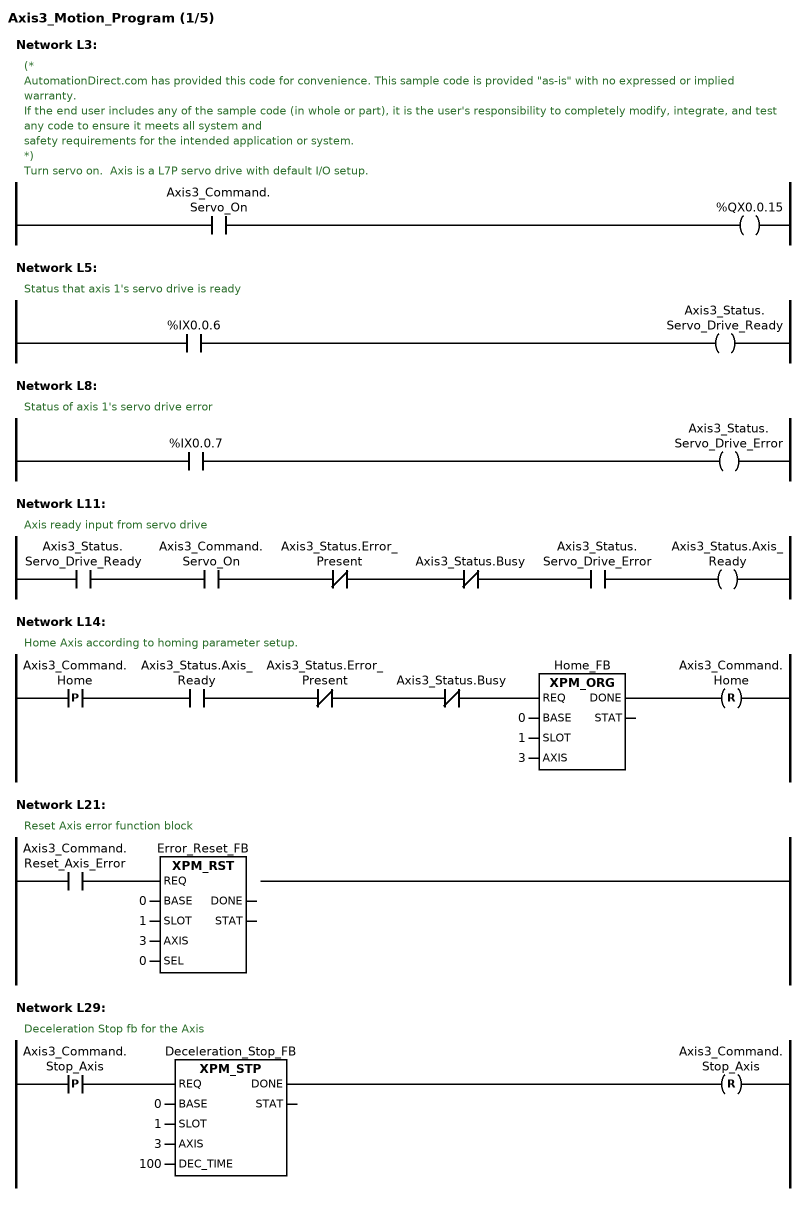
(* ( * / AutomationDirect.com has provided this code for convenience. This sample code is provided "as-is" with no expressed or implied warranty. / If the end user includes any of the sample code (in whole or part), it is the user's responsibility to completely modify, integrate, and test any code to ensure it meets all system and / safety requirements for the intended application or system. / * ) *)
(* Turn servo on.  Axis is a L7P servo drive with default I/O setup. *)
(* Rung L3 *)
%QX0.0.15 := Axis3_Command.Servo_On;
(* Status that axis 1's servo drive is ready *)
(* Rung L5 *)
Axis3_Status.Servo_Drive_Ready := %IX0.0.6;
(* Status of axis 1's servo drive error *)
(* Rung L8 *)
Axis3_Status.Servo_Drive_Error := %IX0.0.7;
(* Axis ready input from servo drive *)
(* Rung L11 *)
Axis3_Status.Axis_Ready := Axis3_Status.Servo_Drive_Ready AND Axis3_Command.Servo_On AND NOT Axis3_Status.Error_Present AND NOT Axis3_Status.Busy AND Axis3_Status.Servo_Drive_Error;
(* Home Axis according to homing parameter setup. *)
(* Rung L14 *)
_e1(CLK := Axis3_Command.Home);
Home_FB(REQ := _e1.Q AND Axis3_Status.Axis_Ready AND NOT Axis3_Status.Error_Present AND NOT Axis3_Status.Busy, BASE := 0, SLOT := 1, AXIS := 3);
IF Home_FB.DONE THEN Axis3_Command.Home := FALSE; END_IF;
(* Reset Axis error function block *)
(* Rung L21 *)
Error_Reset_FB(REQ := Axis3_Command.Reset_Axis_Error, BASE := 0, SLOT := 1, AXIS := 3, SEL := 0);
(* Deceleration Stop fb for the Axis *)
(* Rung L29 *)
_e2(CLK := Axis3_Command.Stop_Axis);
Deceleration_Stop_FB(REQ := _e2.Q, BASE := 0, SLOT := 1, AXIS := 3, DEC_TIME := 100);
IF Deceleration_Stop_FB.DONE THEN Axis3_Command.Stop_Axis := FALSE; END_IF;

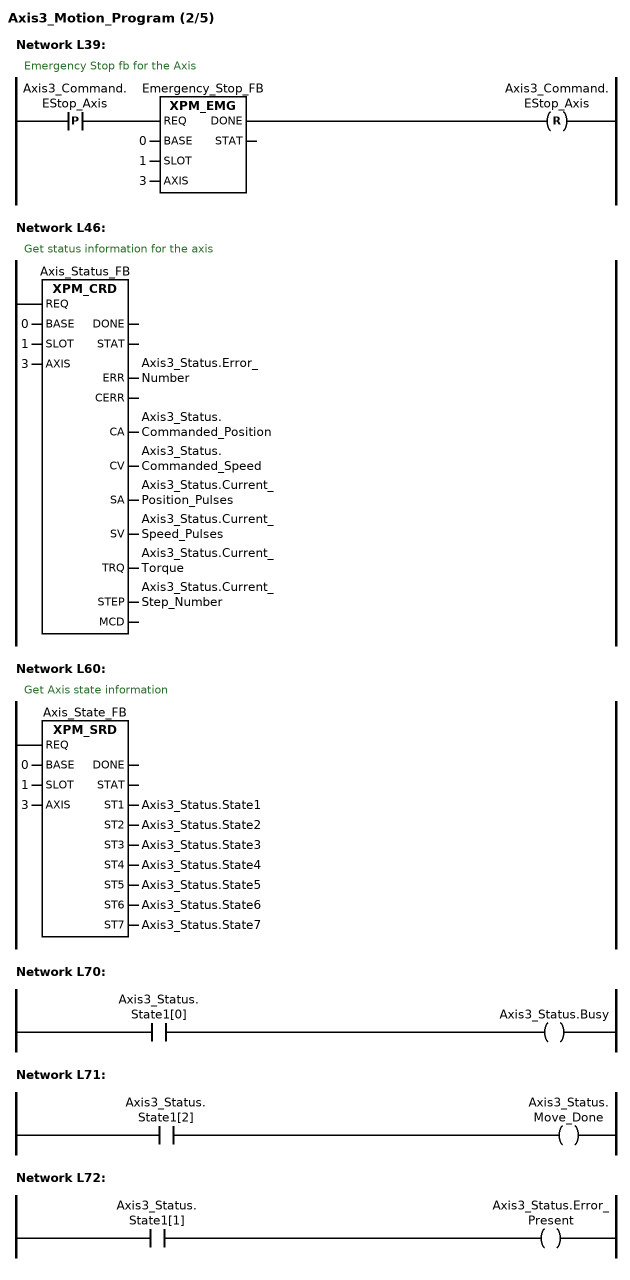
(* Emergency Stop fb for the Axis *)
(* Rung L39 *)
_e3(CLK := Axis3_Command.EStop_Axis);
Emergency_Stop_FB(REQ := _e3.Q, BASE := 0, SLOT := 1, AXIS := 3);
IF Emergency_Stop_FB.DONE THEN Axis3_Command.EStop_Axis := FALSE; END_IF;
(* Get status information for the axis *)
(* Rung L46 *)
Axis_Status_FB(REQ := TRUE, BASE := 0, SLOT := 1, AXIS := 3, ERR => Axis3_Status.Error_Number, CA => Axis3_Status.Commanded_Position, CV => Axis3_Status.Commanded_Speed, SA => Axis3_Status.Current_Position_Pulses, SV => Axis3_Status.Current_Speed_Pulses, TRQ => Axis3_Status.Current_Torque, STEP => Axis3_Status.Current_Step_Number);
(* Get Axis state information *)
(* Rung L60 *)
Axis_State_FB(REQ := TRUE, BASE := 0, SLOT := 1, AXIS := 3, ST1 => Axis3_Status.State1, ST2 => Axis3_Status.State2, ST3 => Axis3_Status.State3, ST4 => Axis3_Status.State4, ST5 => Axis3_Status.State5, ST6 => Axis3_Status.State6, ST7 => Axis3_Status.State7);
(* Rung L70 *)
Axis3_Status.Busy := Axis3_Status.State1[0];
(* Rung L71 *)
Axis3_Status.Move_Done := Axis3_Status.State1[2];
(* Rung L72 *)
Axis3_Status.Error_Present := Axis3_Status.State1[1];

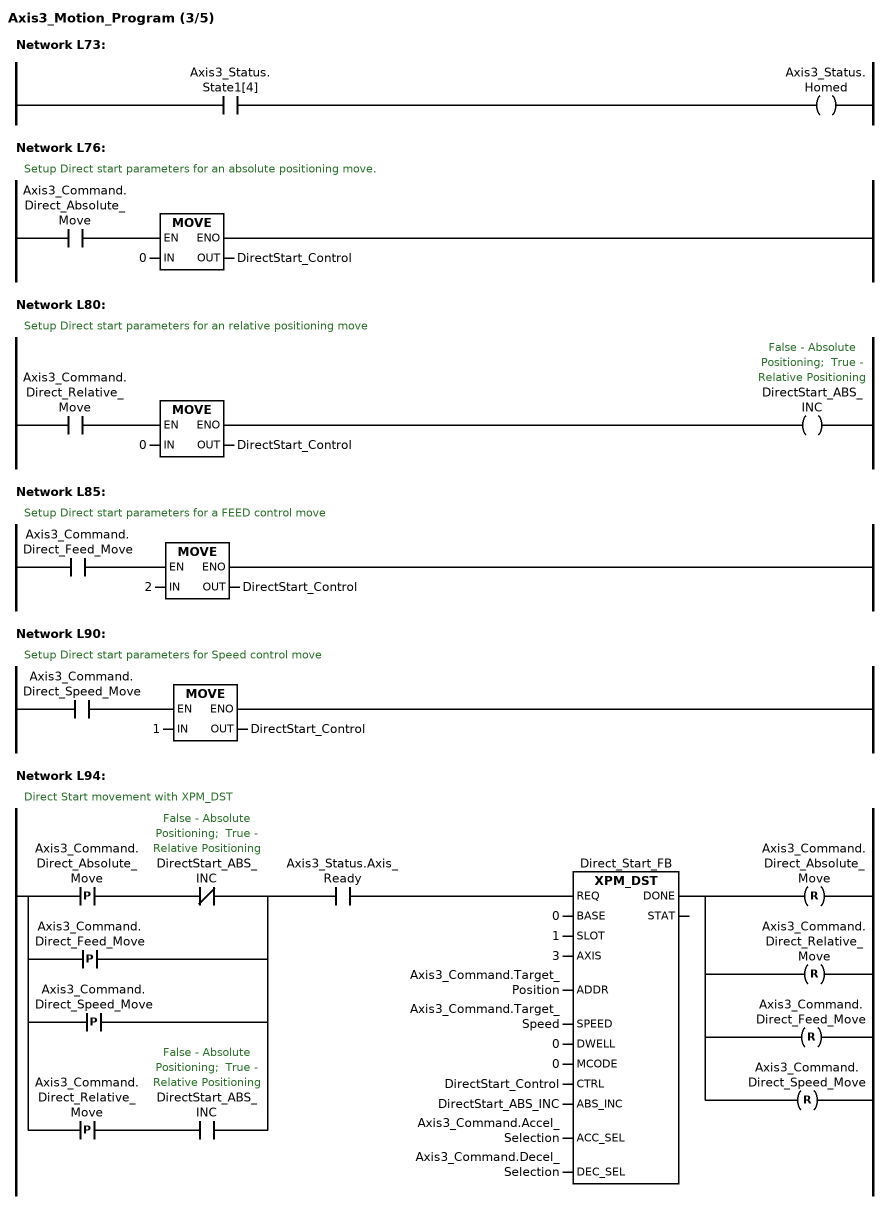
(* Rung L73 *)
Axis3_Status.Homed := Axis3_Status.State1[4];
(* Setup Direct start parameters for an absolute positioning move. *)
(* Rung L76 *)
IF Axis3_Command.Direct_Absolute_Move THEN DirectStart_Control := 0; END_IF;
(* Setup Direct start parameters for an relative positioning move *)
(* Rung L80 *)
IF Axis3_Command.Direct_Relative_Move THEN DirectStart_Control := 0; END_IF;
DirectStart_ABS_INC := Axis3_Command.Direct_Relative_Move;
(* Setup Direct start parameters for a FEED control move *)
(* Rung L85 *)
IF Axis3_Command.Direct_Feed_Move THEN DirectStart_Control := 2; END_IF;
(* Setup Direct start parameters for Speed control move *)
(* Rung L90 *)
IF Axis3_Command.Direct_Speed_Move THEN DirectStart_Control := 1; END_IF;
(* Direct Start movement with XPM_DST *)
(* Rung L94 *)
_e4(CLK := Axis3_Command.Direct_Absolute_Move);
_e5(CLK := Axis3_Command.Direct_Feed_Move);
_e6(CLK := Axis3_Command.Direct_Speed_Move);
_e7(CLK := Axis3_Command.Direct_Relative_Move);
Direct_Start_FB(REQ := ((_e4.Q AND NOT DirectStart_ABS_INC) OR _e5.Q OR _e6.Q OR (_e7.Q AND DirectStart_ABS_INC)) AND Axis3_Status.Axis_Ready, BASE := 0, SLOT := 1, AXIS := 3, ADDR := Axis3_Command.Target_Position, SPEED := Axis3_Command.Target_Speed, DWELL := 0, MCODE := 0, CTRL := DirectStart_Control, ABS_INC := DirectStart_ABS_INC, ACC_SEL := Axis3_Command.Accel_Selection, DEC_SEL := Axis3_Command.Decel_Selection);
IF Direct_Start_FB.DONE THEN
    Axis3_Command.Direct_Absolute_Move := FALSE;
    Axis3_Command.Direct_Relative_Move := FALSE;
    Axis3_Command.Direct_Feed_Move := FALSE;
    Axis3_Command.Direct_Speed_Move := FALSE;
END_IF;

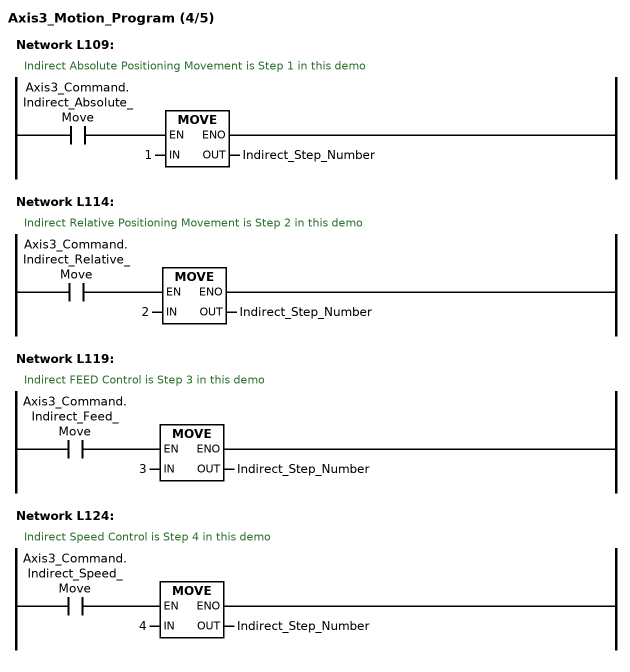
(* Indirect Absolute Positioning Movement is Step 1 in this demo *)
(* Rung L109 *)
IF Axis3_Command.Indirect_Absolute_Move THEN Indirect_Step_Number := 1; END_IF;
(* Indirect Relative Positioning Movement is Step 2 in this demo *)
(* Rung L114 *)
IF Axis3_Command.Indirect_Relative_Move THEN Indirect_Step_Number := 2; END_IF;
(* Indirect FEED Control is Step 3 in this demo *)
(* Rung L119 *)
IF Axis3_Command.Indirect_Feed_Move THEN Indirect_Step_Number := 3; END_IF;
(* Indirect Speed Control is Step 4 in this demo *)
(* Rung L124 *)
IF Axis3_Command.Indirect_Speed_Move THEN Indirect_Step_Number := 4; END_IF;

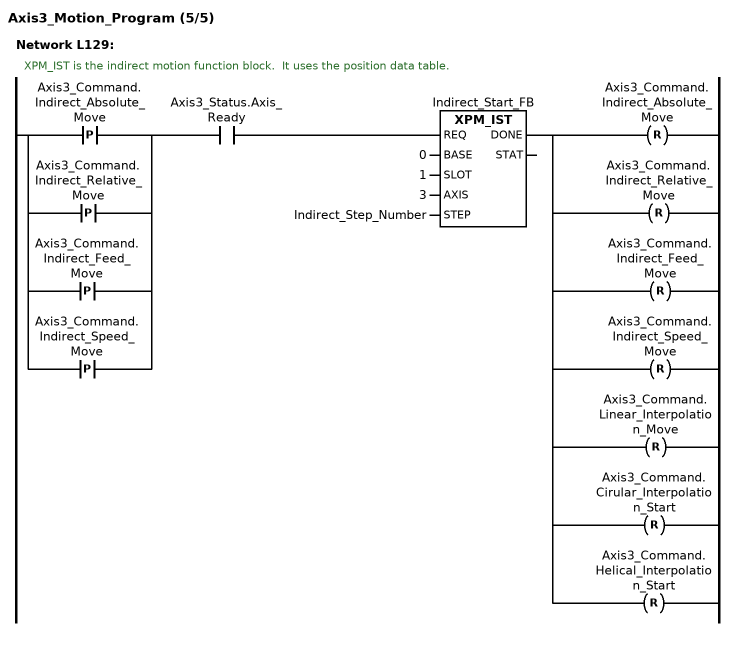
(* XPM_IST is the indirect motion function block.  It uses the position data table. *)
(* Rung L129 *)
_e8(CLK := Axis3_Command.Indirect_Absolute_Move);
_e9(CLK := Axis3_Command.Indirect_Relative_Move);
_e10(CLK := Axis3_Command.Indirect_Feed_Move);
_e11(CLK := Axis3_Command.Indirect_Speed_Move);
Indirect_Start_FB(REQ := (_e8.Q OR _e9.Q OR _e10.Q OR _e11.Q) AND Axis3_Status.Axis_Ready, BASE := 0, SLOT := 1, AXIS := 3, STEP := Indirect_Step_Number);
IF Indirect_Start_FB.DONE THEN
    Axis3_Command.Indirect_Absolute_Move := FALSE;
    Axis3_Command.Indirect_Relative_Move := FALSE;
    Axis3_Command.Indirect_Feed_Move := FALSE;
    Axis3_Command.Indirect_Speed_Move := FALSE;
    Axis3_Command.Linear_Interpolation_Move := FALSE;
    Axis3_Command.Cirular_Interpolation_Start := FALSE;
    Axis3_Command.Helical_Interpolation_Start := FALSE;
END_IF;
END_PROGRAM

PROGRAM XPM_SST_DEMO (* task: Scan Program *)
VAR
    INST1 : XPM_SST;
    SST_Axis : USINT; (* choose which axes run with the XPM_SST *)
    StartSST : BOOL; (* start the XPM_SST program. *)
END_VAR

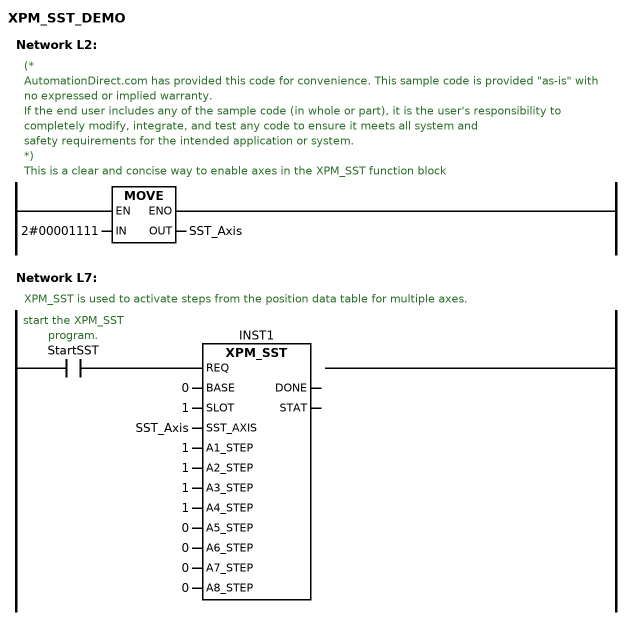
(* ( * / AutomationDirect.com has provided this code for convenience. This sample code is provided "as-is" with no expressed or implied warranty. / If the end user includes any of the sample code (in whole or part), it is the user's responsibility to completely modify, integrate, and test any code to ensure it meets all system and / safety requirements for the intended application or system. / * ) *)
(* This is a clear and concise way to enable axes in the XPM_SST function block *)
(* Rung L2 *)
SST_Axis := 2#00001111;
(* XPM_SST is used to activate steps from the position data table for multiple axes. *)
(* Rung L7 *)
INST1(REQ := StartSST, BASE := 0, SLOT := 1, SST_AXIS := SST_Axis, A1_STEP := 1, A2_STEP := 1, A3_STEP := 1, A4_STEP := 1, A5_STEP := 0, A6_STEP := 0, A7_STEP := 0, A8_STEP := 0);
END_PROGRAM

PROGRAM Servo_Control (* task: Scan Program *)
(* Commands for turning on servos and acknowledging alarms *)
VAR_EXTERNAL
    Axis1_Command : Motion_Command_type; (* Commands for Axis 1 *)
    Axis2_Command : Motion_Command_type; (* Commands for Axis 2 *)
    Axis3_Command : Motion_Command_type; (* Commands for Axis 3 *)
    Reset_Servo_Errors : BOOL; (* Acknowledge servo errors *)
    Turn_On_Servos : BOOL; (* Command to turn on all the servos *)
END_VAR

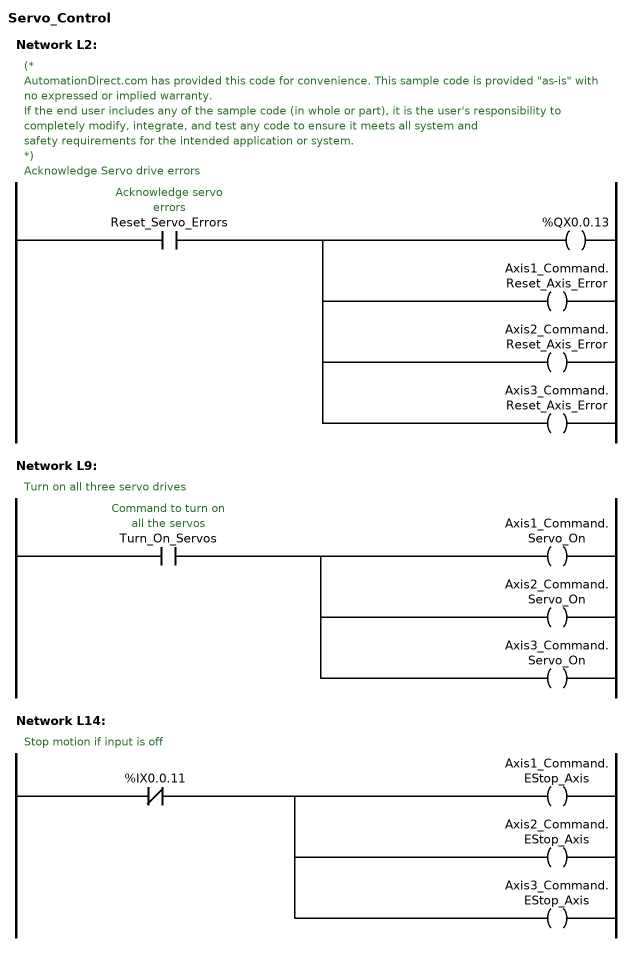
(* ( * / AutomationDirect.com has provided this code for convenience. This sample code is provided "as-is" with no expressed or implied warranty. / If the end user includes any of the sample code (in whole or part), it is the user's responsibility to completely modify, integrate, and test any code to ensure it meets all system and / safety requirements for the intended application or system. / * ) *)
(* Acknowledge Servo drive errors *)
(* Rung L2 *)
%QX0.0.13 := Reset_Servo_Errors;
Axis1_Command.Reset_Axis_Error := Reset_Servo_Errors;
Axis2_Command.Reset_Axis_Error := Reset_Servo_Errors;
Axis3_Command.Reset_Axis_Error := Reset_Servo_Errors;
(* Turn on all three servo drives *)
(* Rung L9 *)
Axis1_Command.Servo_On := Turn_On_Servos;
Axis2_Command.Servo_On := Turn_On_Servos;
Axis3_Command.Servo_On := Turn_On_Servos;
(* Stop motion if input is off *)
(* Rung L14 *)
Axis1_Command.EStop_Axis := NOT %IX0.0.11;
Axis2_Command.EStop_Axis := NOT %IX0.0.11;
Axis3_Command.EStop_Axis := NOT %IX0.0.11;
END_PROGRAM